/// cyclically reads the  cpu temp at specified update period. Default is 500ms.
{attribute 'contains_implicit_enum'}
FUNCTION_BLOCK T_MdpReadCpuTemp
VAR
   /// local read                
   amsNetId : STRING := '';
   mdpAddr : ST_MDP_Addr;
   updateTimer : TON := (PT := TIME#500ms);
   readMdpElement : FB_MDP_ReadElement;
   /// returned from MDP read element 
   rawData : UINT;
   _cpuTemp : INT;
   {attribute 'implicit_enum_type' := ''}
   state : (
      mrctInit := 0, // initiate state machine (set parameters)
      mrctReadCpuTemp,
      mrctWaitForReadComplete,
      mrctProcessCpuTemp
   );
END_VAR
VAR CONSTANT
   /// from IPC Diagnostics Manual V1.8, p63 
   CPU_PROPERTIES_TABLE_NUMBER : BYTE := 1;
   /// from IPC Diagnostics Manual V1.8, p63 
   CPU_TEMP_SUB_INDEX_OF_CPU_PROPS_TABLE : BYTE := 3;
END_VAR

CASE state OF

   mrctInit:

      // timer starts the read process.
      state :=
         SEL(updateTimer.Q, state, mrctReadCpuTemp);

   mrctReadCpuTemp:

      state := mrctWaitForReadComplete;

   mrctWaitForReadComplete:

      IF NOT readMdpElement.bBusy THEN

         state := mrctProcessCpuTemp;

      END_IF

   mrctProcessCpuTemp:

      IF NOT readMdpElement.bError THEN
         MEMCPY(ADR(_cpuTemp), ADR(rawData), SIZEOF(rawData));

      END_IF

      state := mrctInit;

ELSE

   state := mrctInit;

END_CASE

updateTimer(
   IN := state = mrctInit
);

mdpAddr.nArea := INT_TO_BYTE(eMDP_Area_ConfigArea);
mdpAddr.nTableId := CPU_PROPERTIES_TABLE_NUMBER;
mdpAddr.nSubIdx := CPU_TEMP_SUB_INDEX_OF_CPU_PROPS_TABLE;

readMdpElement(
   bExecute := state = mrctReadCpuTemp,
   eModuleType := E_MDP_ModuleType.eMDP_ModT_CPU,
   stMDP_Addr := mdpAddr,
   iModIdx := 0,
   pDstBuf := ADR(rawData),
   cbDstBufLen := SIZEOF(rawData),
   sAmsNetId := amsNetId,
);

{attribute 'monitoring' := 'variable'}
PROPERTY Busy : BOOL
GET
Busy := state <> mrctInit;
END_GET
END_PROPERTY

{attribute 'monitoring' := 'call'}
PROPERTY CpuTemp : INT
GET
CpuTemp := THIS^._cpuTemp;
END_GET
END_PROPERTY

{attribute 'monitoring' := 'variable'}
PROPERTY Error : BOOL
GET
Error := NOT Busy AND readMdpElement.bError;
END_GET
END_PROPERTY

{attribute 'monitoring' := 'variable'}
PROPERTY ErrorId : UDINT
GET
ErrorId := SEL(Busy, readMdpElement.nErrID, 0);
END_GET
END_PROPERTY

METHOD SetUpdateTimerValue
VAR_INPUT
   UpdatePeriod : TIME;
END_VAR
IF UpdatePeriod > T#1MS THEN
   THIS^.updateTimer.PT := UpdatePeriod;
END_IF
END_METHOD

END_FUNCTION_BLOCK

(* stored: Version 1.1.0.1, ProductVersion 3.1.4024.9
   POU T_MdpReadCpuTemp: Id {e0065e76-d33a-4e1b-a8bc-52fca8279681}, SpecialFunc None
   Property Busy: Id {fdefc8c5-2d51-4f3f-b7dc-6050cfc8022e}
   Get Get: Id {1f2eec0b-628f-46de-b9c3-8e6ef8fa80e3}
   Property CpuTemp: Id {8825d759-f03d-458c-b53d-c4b34db13039}
   Get Get: Id {849c0c14-513d-4cad-9600-70f382d07c9a}
   Property Error: Id {b377bdf0-eee3-4f8a-8532-1a443c8d6e90}
   Get Get: Id {146efe53-e3fc-4f51-aa4d-8a47191b0902}
   Property ErrorId: Id {71f8c472-e21b-4090-a549-ebb9bfb87bc1}
   Get Get: Id {416a38a4-c638-4f00-a26b-9c06c0826534}
   Method SetUpdateTimerValue: Id {ec3d15a0-c102-46bf-a9be-641e6336c5c8} *)
